FUNCTION_BLOCK FB_System_AKM_941
VAR_INPUT
	Freigabe_auto			: BOOL;
	Betrieb_Anford_auto		: BOOL;
	Regelung_Modus_auto		: SINT;
	Regelung_Sollw_auto		: REAL;
END_VAR
VAR_OUTPUT
	{attribute 'OPC.UA.DA' := '1'}Steuerung				: ST_System_AKM_Steuerung;		
	{attribute 'OPC.UA.DA' := '1'}Stellwert				: ST_System_AKM_Stellwert;		
	{attribute 'OPC.UA.DA' := '1'}Zustand					: ST_System_AKM_Zustand;	
	{attribute 'OPC.UA.DA' := '1'}Parameter				: ST_System_AKM_Parameter;		
END_VAR
VAR
	Zustandscheck			: FB_System_AKM_Zustandscheck;
	Logik					: FB_System_AKM_Logik;
	Ablaufsteuerung			: FB_System_AKM_Ablaufsteuerung;
	Sollwertscheck			: FB_System_AKM_Sollwertscheck;
	Regelung				: FB_System_AKM_Regelung;
	Stellwertscheck			: FB_System_AKM_Stellwertscheck;

	AKM_941					: FB_AKM;
	AKM_941_Zuweisung		: FB_AKM_Zuweisung;
END_VAR

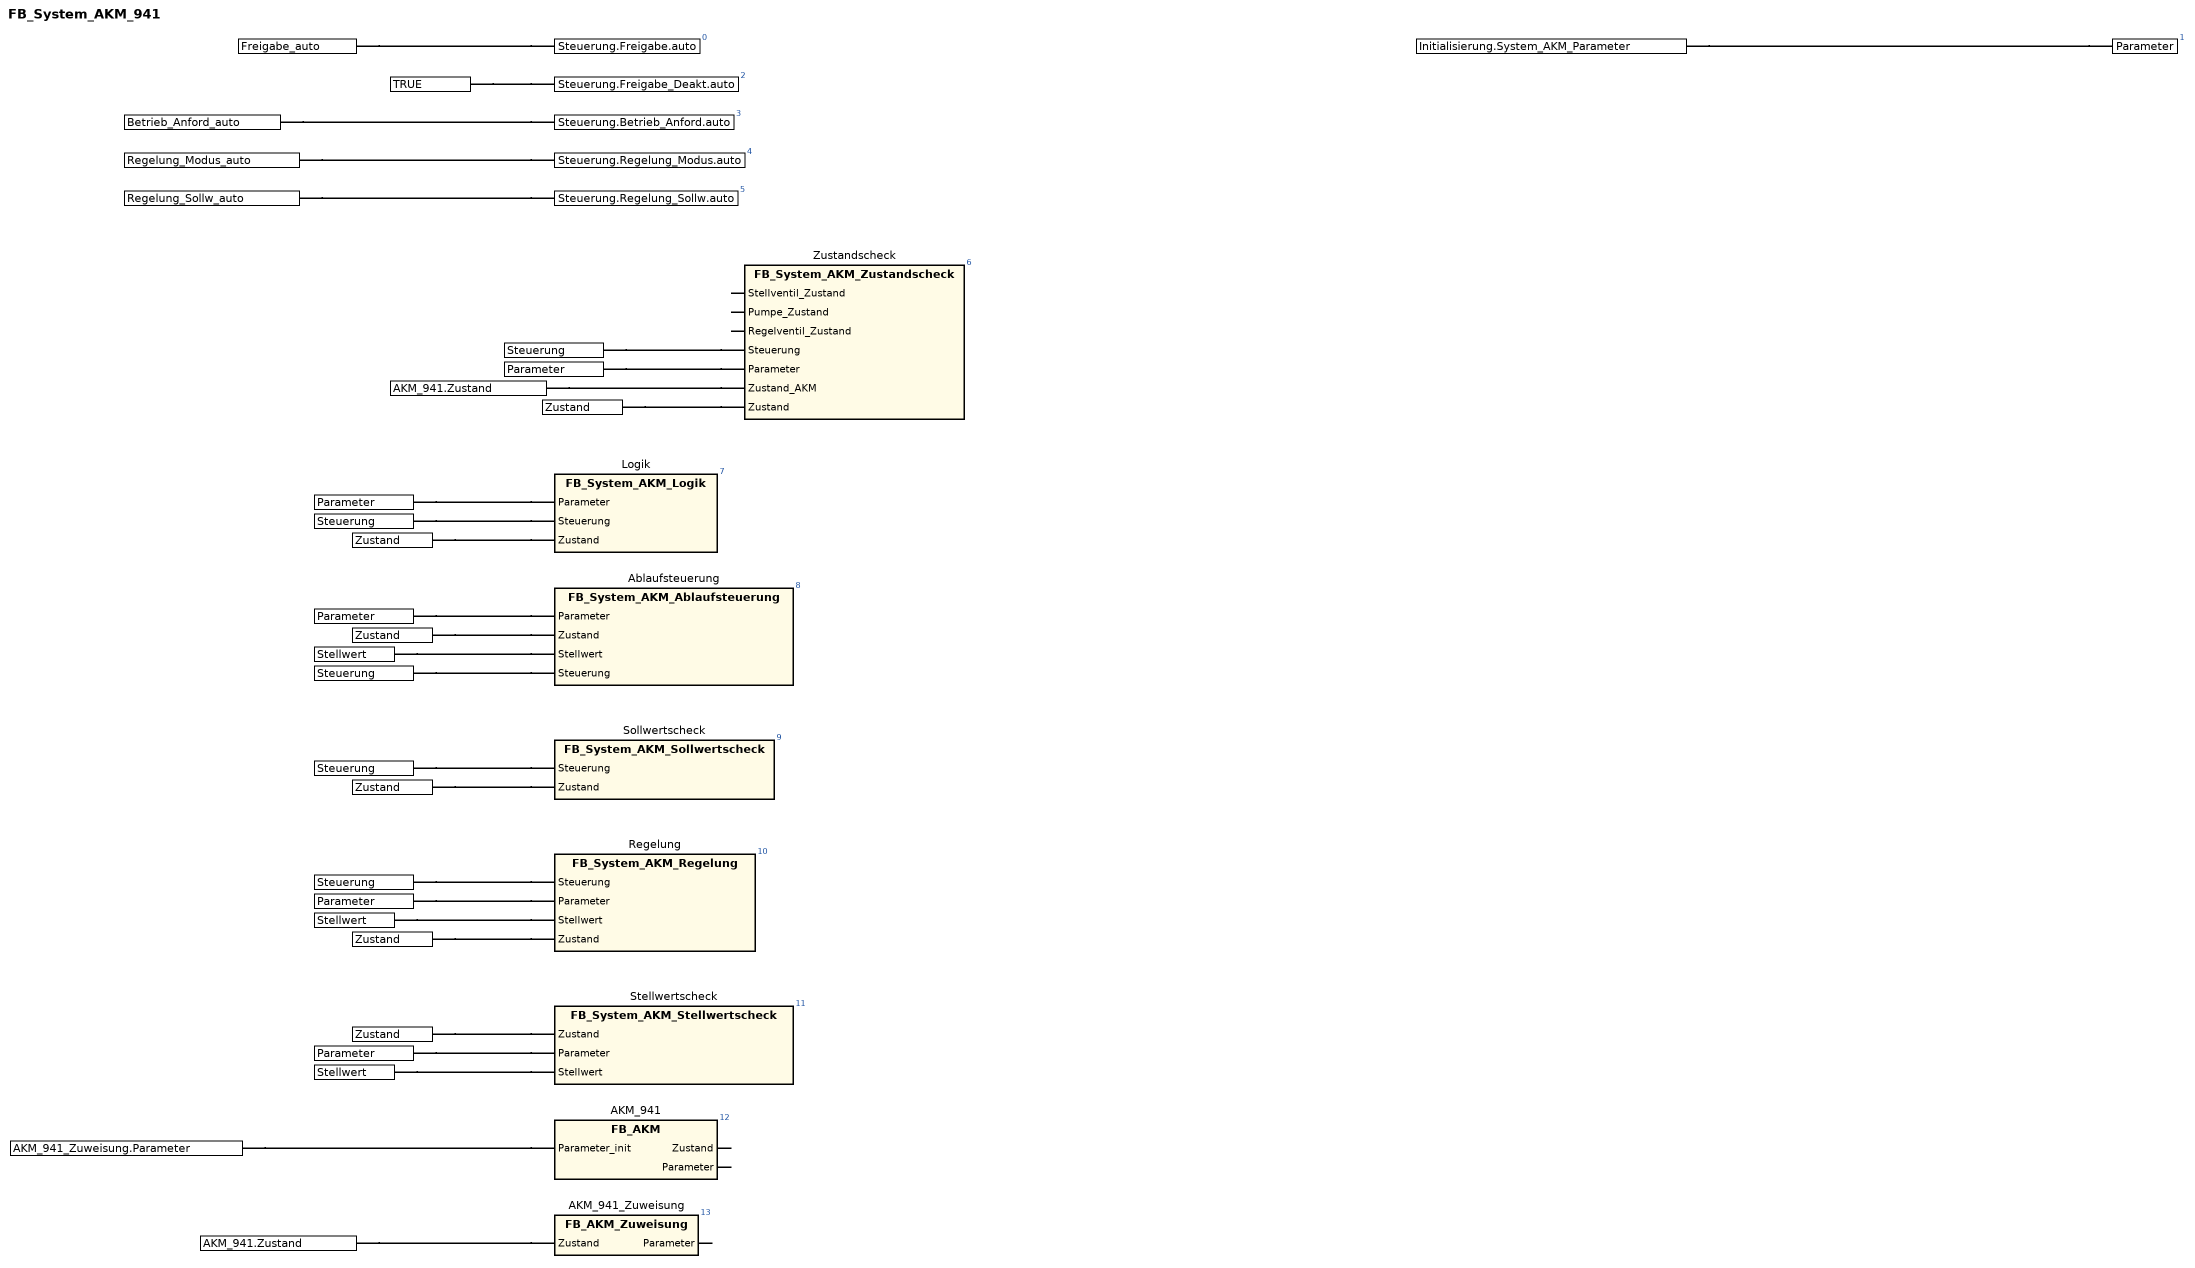
Steuerung.Freigabe.auto := Freigabe_auto;
Parameter := Initialisierung.System_AKM_Parameter;
Steuerung.Freigabe_Deakt.auto := TRUE;
Steuerung.Betrieb_Anford.auto := Betrieb_Anford_auto;
Steuerung.Regelung_Modus.auto := Regelung_Modus_auto;
Steuerung.Regelung_Sollw.auto := Regelung_Sollw_auto;
Zustandscheck(
    Steuerung := Steuerung,
    Parameter := Parameter,
    Zustand_AKM := AKM_941.Zustand,
    Zustand := Zustand); // FB_System_AKM_Zustandscheck
Logik(Parameter := Parameter, Steuerung := Steuerung, Zustand := Zustand); // FB_System_AKM_Logik
Ablaufsteuerung(Parameter := Parameter, Zustand := Zustand, Stellwert := Stellwert, Steuerung := Steuerung); // FB_System_AKM_Ablaufsteuerung
Sollwertscheck(Steuerung := Steuerung, Zustand := Zustand); // FB_System_AKM_Sollwertscheck
Regelung(Steuerung := Steuerung, Parameter := Parameter, Stellwert := Stellwert, Zustand := Zustand); // FB_System_AKM_Regelung
Stellwertscheck(Zustand := Zustand, Parameter := Parameter, Stellwert := Stellwert); // FB_System_AKM_Stellwertscheck
AKM_941(Parameter_init := AKM_941_Zuweisung.Parameter); // FB_AKM
AKM_941_Zuweisung(Zustand := AKM_941.Zustand); // FB_AKM_Zuweisung

END_FUNCTION_BLOCK

(* stored: Version 1.1.0.1, ProductVersion 3.1.4024.9
   POU FB_System_AKM_941: Id {dd388b55-a4ab-4a93-ae62-24136e3c4fab}, SpecialFunc None *)
